FUNCTION F_Add : INT
VAR_INPUT
		iValue : INT;
END_VAR
VAR
END_VAR

//iValue := iValue + 10;
F_Add :=  iValue +  10;


(*iNumber remains 5 Because function modified only copy *)

END_FUNCTION

(* stored: Version 1.1.0.1, ProductVersion 3.1.4024.16
   POU F_Add: Id {795e5762-f6ee-4d3d-b93c-a8f107056e8a}, SpecialFunc None *)
